// TIA Portal V18 export
FUNCTION "_hmi_main" : Void   // FC26, FBD
{ S7_Optimized_Access := 'TRUE' }
VERSION : 0.1
// stored: AutoNumber true, IsIECCheckEnabled false, SetENOAutomatically false, UDAEnableTagReadback false
BEGIN

REGION Network 1
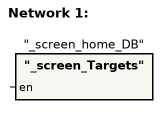
   "_screen_home_DB"();   // "_screen_Targets"
END_REGION
END_FUNCTION
